// Mitsubishi GX Works2 project: COUNTER_EX   PLC: Q03UDV

PROGRAM MAIN
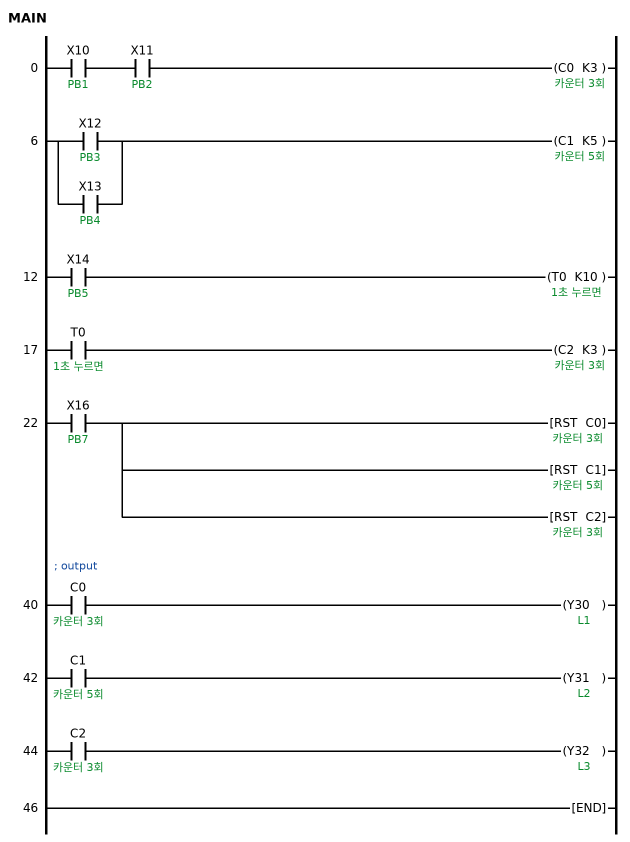
0     LD      X10  ; PB1
      AND     X11  ; PB2
      OUT     C0 K3  ; 카운터 3회
6     LD      X12  ; PB3
      OR      X13  ; PB4
      OUT     C1 K5  ; 카운터 5회
12    LD      X14  ; PB5
      OUT     T0 K10  ; 1초 누르면
17    LD      T0  ; 1초 누르면
      OUT     C2 K3  ; 카운터 3회
22    LD      X16  ; PB7
      RST     C0  ; 카운터 3회
      RST     C1  ; 카운터 5회
      RST     C2  ; 카운터 3회
; output
40    LD      C0  ; 카운터 3회
      OUT     Y30  ; L1
42    LD      C1  ; 카운터 5회
      OUT     Y31  ; L2
44    LD      C2  ; 카운터 3회
      OUT     Y32  ; L3
46    END
END_PROGRAM
